{attribute 'qualified_only'}
{attribute 'strict'}
TYPE  E_WashProgram :
(
	NONE         := 0,
    SOFT      := 1,
    NORMAL    := 2,
    HEAVY     := 3
);
END_TYPE

(* stored: Version 1.1.0.1, ProductVersion 3.1.4024.16
   DUT E_WashProgram: Id {e27fb257-593f-41d4-9eda-27412b1347c9} *)
